FUNCTION_BLOCK TLController (* Composite Function Block Type *)
  (* Standard: 61499-2 *)
  (* Version 0.2, 2003-12-05, JHC, Rockwell Automation, Renamed from NEWCOMPFB. *)
  (* Version 0.1, 2002-01-08, JHC, Rockwell Automation, Added DLY FB as example. *)
  (* Version 0.0, 2000-05-27, JHC, Rockwell Automation *)
  (* Compiler header: package fb.rt.template; *)
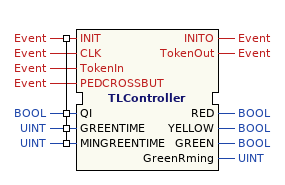
  EVENT_INPUT
    INIT WITH QI, GREENTIME, MINGREENTIME; (* Initialization Request *)
    CLK;
    TokenIn;
    PEDCROSSBUT;
  END_EVENT
  EVENT_OUTPUT
    INITO; (* Initialization Confirm *)
    TokenOut;
  END_EVENT
  VAR_INPUT
    QI : BOOL; (* Input event qualifier *)
    GREENTIME : UINT;
    MINGREENTIME : UINT;
  END_VAR
  VAR_OUTPUT
    RED : BOOL;
    YELLOW : BOOL;
    GREEN : BOOL;
    GreenRming : UINT;
  END_VAR
  FBS
    ButPressCTR : E_CTU(PV := 4);
    Controller : Controller;
  END_FBS
  EVENT_CONNECTIONS
    PEDCROSSBUT TO ButPressCTR.CU;
    INIT TO Controller.INIT;
    CLK TO Controller.CLK;
  END_CONNECTIONS
  DATA_CONNECTIONS
    GreenRming TO Controller.GREENTIME;
    ButPressCTR.Q TO Controller.PEDCROSS;
  END_CONNECTIONS
END_FUNCTION_BLOCK
